// TIA Portal V17 export
// export: Created 2024-09-02T12:50:07.6727563Z, ExportSetting WithDefaults, DisplayName Totally Integrated Automation Portal, DisplayVersion V17, DisplayName TIA Portal Openness, DisplayVersion V17, DisplayName TIA Portal Version Control Interface, DisplayVersion V17, DisplayName STEP 7 Professional, DisplayVersion V17, DisplayName STEP 7 Safety, DisplayVersion V17, DisplayName WinCC Professional, DisplayVersion V17
DATA_BLOCK "GraDB2_FG01_Station_OP70"   // DB1262
{ S7_Optimized_Access := 'TRUE'; DB_Accessible_From_OPC_UA := 'FALSE' }
AUTHOR : VAF
FAMILY : SK
NAME : SK
VERSION : 0.1
// stored: AutoNumber false, DBAccessibleFromOPCUA false, IsOnlyStoredInLoadMemory false, IsRetainMemResEnabled false, IsWriteProtectedInAS false, MemoryReserve 0
   VAR
      Home { ExternalWritable := 'False'} : Bool;   // Grundstellung
      Home_Mechanic { ExternalWritable := 'False'} : Bool;   // Grundstellung Mechanik / Basic position mechanic
      Home_SQ { ExternalWritable := 'False'} : Bool;   // Grundstellung Schrittkette / Basic position Step chain
      Finished { ExternalWritable := 'False'} : Bool := false;   // Fertigmeldung / Finished message
      Finished_OK : Bool;
      Finished_NOK : Bool;
      Finished_Reset { ExternalWritable := 'False'} : Bool;   // Fertigmeldung Reset / Finished Reset
      SQ_Finished { ExternalWritable := 'False'} : Bool;   // Ablauf Schrittkette fertig / Sequence cycle finished
      Workers { ExternalWritable := 'False'; S7_SetPoint := 'True'} : "TypeSKS_OPERATOR";   // Schrittmerker / Step marker
      "MM110 Sliding Damper Cap" { S7_SetPoint := 'True'} : "TypeSKS_HORI";
      "MM120 Sliding Ball" { S7_SetPoint := 'True'} : "TypeSKS_HORI";
      "MM130 Press Damper Cap" { S7_SetPoint := 'True'} : "TypeSKS_VERT";
      Proces_Press_active : Bool;
      Proces_Slider_Ball_Active : Bool;
      Proces_Slider_DamperCap_Active : Bool;
      "Feeder Blowing Air On" { S7_SetPoint := 'True'} : "TypeSKS_Feeder_Unit";
      Feeder_Damper_Cap : Struct
         "A" : Struct
            on : Bool;
            off : Bool;
            Part_Out : Bool;
         END_STRUCT;
         H : Struct
            on : Bool;
            off : Bool;
            R_Part_insite : Bool;
            R_Part_in_Separator : Bool;
            R_Part_in_pipe : Bool;
            S_Part_insite : Bool;
            S_Part_in_Separator : Bool;
            S_Part_in_pipe : Bool;
         END_STRUCT;
         Status : Struct
            Part_insite : Bool;
            Part_in_Separator : Bool;
            Part_in_pipe : Bool;
         END_STRUCT;
      END_STRUCT;
      "MM220 Sliding Separation Cylinder Dumper Cap" { S7_SetPoint := 'True'} : "TypeSKS_HORI";
      "MM210 Loading Cylinder Dumper Cap" { S7_SetPoint := 'True'} : "TypeSKS_VERT";
      "MM210 Loading Cylinder_Work" { S7_SetPoint := 'True'} : Bool;
      Feeder_Ball : Struct
         "A" : Struct
            on : Bool;
            off : Bool;
            Part_Out : Bool;
         END_STRUCT;
         H : Struct
            on : Bool;
            off : Bool;
            R_Part_insite : Bool;
            R_Part_in_Separator : Bool;
            R_Part_in_pipe : Bool;
            S_Part_insite : Bool;
            S_Part_in_Separator : Bool;
            S_Part_in_pipe : Bool;
         END_STRUCT;
         Status : Struct
            Part_insite : Bool;
            Part_in_Separator : Bool;
            Part_in_pipe : Bool;
         END_STRUCT;
      END_STRUCT;
      NIO_Controle : Struct
         HMI_Input : Struct
            X1 : Int;
            X2 : Int;
            Restart : Bool;
         END_STRUCT;
         Staus : Struct
            Warning : Bool;
            Error : Bool;
         END_STRUCT;
         Actual : Struct
            Counter_NOK : IEC_COUNTER;
         END_STRUCT;
      END_STRUCT;
      Uncorrect_Pallet_Position : Bool;
      Retry : Array[1..8] of Struct
         Max_Retry : Int;
         Actual_Retry : Int;
         "Counter" : IEC_COUNTER;
      END_STRUCT;
      fpDamperCap_Feed_Deselection : Bool;
      fnDamperCap_Feed_Deselection : Bool;
   END_VAR
BEGIN
   Retry[1..8].Max_Retry := 2;
END_DATA_BLOCK
